TYPE ST_canRxdata :
STRUCT
	cobID			: STRING;
	deviceID		: ARRAY [1..12] OF STRING; // will make it 1..10 later
	byteData		: ARRAY [0..7] OF USINT;
	byteData_hexstr	: ARRAY [0..7] OF STRING;
END_STRUCT
END_TYPE

(* stored: Version 1.1.0.1, ProductVersion 3.1.4024.11
   DUT ST_canRxdata: Id {e25865d4-bfca-468c-b00c-09aae9848e51} *)
